(*
  Mark camera system on WEU machine
  1 mark sensor (optional: reverse mode - roll printed in reversed direction, sensor moved to other side)
*)
FUNCTION_BLOCK FB_MarkCamera_WEU EXTENDS FB_CameraBase 
VAR_INPUT
END_VAR
VAR
  // config
  _iMarkDefinition          : I_MarkDefinition;
  // helper
  pMark                     : POINTER TO ST_MarkDefinition;
END_VAR

IF NOT _bInitialized THEN RETURN; END_IF

// The detection work is done in FB_CameraDetection
// This FB just uses(receives) the marks from the external implementation
// - Receives events CamTrigger & CamTriggerDone from MarkDetection
// - Get current marks and send them to the iCameraSink

WHILE _iMarkDefinition.nMarksDetected > _nRxCamPoints DO
  
  pMark := _iMarkDefinition.getMark(nIdx:=_nRxCamPoints+1);
  IF pMark <> 0 THEN
    // Send Mark (CamPoint) to CameraSink
    stCamPoint.x_ref := F_MeterToSubPixelReal(  fPosMeter:=pMark^.fPosX                                 (*[m]*)
                                              , fResoSubPx:=UDINT_TO_LREAL(_nPrintUnitResolution));     (*Result should be in pixels*)
    stCamPoint.y_ref := F_MeterToSubPixelReal( fPosMeter:=pMark^.fPosX                                  (*[m]*)
                                              , fResoSubPx:=UDINT_TO_LREAL(_nPrintUnitResolution));     (*Result should be in pixels*)
    stCamPoint.dx    := F_MeterToSubPixelReal( fPosMeter:=pMark^.sState.dx                              (*[m]*)
                                              , fResoSubPx:=UDINT_TO_LREAL(_nPrintUnitResolution));     (*Result should be in pixels*)
    stCamPoint.dy    := F_MeterToSubPixelReal( fPosMeter:=pMark^.sState.dy                              (*[m]*)
                                              , fResoSubPx:=UDINT_TO_LREAL(_nPrintUnitResolution));     (*Result should be in pixels*)
    stCamPoint.valid := pMark^.sState.bSet;
  
    IF _iCameraSink <> 0 THEN
      _iCameraSink.AddCamPoint(sDeformationPoint:=stCamPoint);
    END_IF
    
    _nRxCamPoints := _nRxCamPoints + 1;   // next mark
  END_IF
END_WHILE

METHOD CamTrigger
VAR_INPUT
  bOk             : BOOL;     // trigger is ok
	nPos            : DINT;     // camera triggered position
  nPosDeviation   : DINT;     // camera started deviation
END_VAR
IF NOT _bInitialized THEN RETURN; END_IF

SUPER^.CamTrigger(bOk:=bOk, nPos:=nPos, nPosDeviation:=nPosDeviation);
END_METHOD

METHOD CamTriggerDone
IF NOT _bInitialized THEN RETURN; END_IF

{warning 'Finalize mark handling'}

SUPER^.CamTriggerDone();
END_METHOD

{attribute 'monitoring':='call'}
PROPERTY eCameraMode : E_CameraMode
GET
eCameraMode := _eCameraMode;
IF _eCameraMode = E_CameraMode.Auto THEN
  eCameraMode := E_CameraMode.Live;
END_IF
END_GET
END_PROPERTY

PROPERTY eDeviceType : E_CameraDevice
GET
eDeviceType := E_CameraDevice.PrintMark;
END_GET
END_PROPERTY

METHOD GetCamStatus : BOOL
VAR_OUTPUT
  bConnectionOK  : BOOL;    // Camera connected
  bTeachOk       : BOOL;    // Teach successful
  nTeachedPoints : UDINT;   // Teached points for this job
  nScannedPoints : UDINT;   // Scanned points on current sheet
  bCamStarted    : BOOL;    // Camera trigger is active, cam started
  bCamDone       : BOOL;    // Camera finished on last CT
  bErrors        : ARRAY[1..GVL_Camera.nC_NbCamErrors] OF BOOL;  // generic error flag list
END_VAR
IF _iMarkDefinition = 0 THEN RETURN; END_IF

bConnectionOK  := TRUE;
bTeachOk       := (_iMarkDefinition.nMarks > 0);
nTeachedPoints := _iMarkDefinition.nMarks;  // teach marks
nScannedPoints := _nRxCamPoints;
bCamStarted    := _bCamTriggerStarted;
bCamDone       := _bCamTriggerDone;

GetCamStatus := bConnectionOK AND bTeachOk;   // camera ready
END_METHOD

METHOD InitMarkCamera
VAR_INPUT
  nPrintUnitResolution         : UDINT;    (*printhead pixel resolution [dpi]*)
  nPrintUnitSubPx              : UDINT;    (*print unit subPixel resolution [SubPx]*)
  iCameraTrigger               : I_CameraTrigger;
  iMarkDefinition              : I_MarkDefinition;  // mark detection fb
END_VAR
VAR
  bOK : BOOL;
END_VAR
SUPER^.Init( nPrintUnitResolution      := nPrintUnitResolution
           , nPrintUnitSubPx           := nPrintUnitSubPx
           , iCameraTrigger            := iCameraTrigger
           , bUseCameraTrigger         := FALSE
           , bUseCameraTriggerFeedback := FALSE);

IF NOT _bInitialized OR iMarkDefinition = 0 THEN LogError('Init: invalid parameter'); RETURN; END_IF

_iMarkDefinition := iMarkDefinition;

_bInitialized := TRUE;
END_METHOD

METHOD mJobStart : BOOL
IF eCameraMode <> E_CameraMode.NoCorrection THEN TeachMarks(); END_IF
END_METHOD

(*
  Set mode to camera.
  :return: TRUE if success
*)
METHOD setCameraMode : BOOL
VAR_INPUT
  eCameraMode : E_CameraMode;
END_VAR
IF eCameraMode = E_CameraMode.Auto OR
   eCameraMode = E_CameraMode.NoCorrection OR
   eCameraMode = E_CameraMode.Live
   //eCameraMode = E_CameraMode.Trend 
THEN
   
  _eCameraMode := eCameraMode;  // set desired mode
  setCameraMode := TRUE;
ELSE
  LogError(F_Concat3('Camera mode=', TO_STRING(eCameraMode), ' not supported by camera'));
  _eCameraMode := E_CameraMode.NoCorrection;
END_IF
END_METHOD

{attribute 'monitoring':='variable'}
PROPERTY sName : STRING
GET
sName := 'Printmarks';
END_GET
END_PROPERTY

(*
  Calculate marks (position, shape) and register to mark definition. 
*)
METHOD PUBLIC TeachMarks : BOOL
VAR_INPUT
END_VAR
VAR
  i : UDINT;
  spacing : LREAL := 0.08;  // mark spacing
  asq : LREAL := 0.002;     // sqare a length
  atr : LREAL := 0.008;     // triangle length (same h / l)
  numMarks : UDINT;
  xOfs : LREAL := 0.0023;
  yOfs : LREAL := 0.0023;
  
  sNewMark : ST_MarkDefinition;
END_VAR


// TODO: this is only a reference caluclation for simulation, please adpat after definition by STAG
//       ...
IF _iMarkDefinition = 0 THEN RETURN; END_IF

_iMarkDefinition.ResetDefinition();

numMarks := TO_UDINT((_fSubstrateLength-2*xOfs) / spacing); //  // TO_UDINT(FLOOR(_fSubstrateLength / spacing);)
IF numMarks = 0 THEN numMarks := 1; END_IF   // at least one mark

// calculate position
FOR i:=1 TO numMarks DO
  sNewMark.fHeight := atr;
  sNewMark.fTrLength := atr;
  sNewMark.fSqLength := SEL(i>1, asq+1.5*atr, asq);
  sNewMark.fPosX := xOfs+(i-1)*spacing;
  sNewMark.fPosY := yOfs;
  sNewMark.bInvertedX := FALSE;
  
  _iMarkDefinition.RegisterMark(sMark:=sNewMark);
END_FOR
END_METHOD

END_FUNCTION_BLOCK

(* stored: Version 1.1.0.1, ProductVersion 3.1.4024.11
   POU FB_MarkCamera_WEU: Id {022ae170-1450-4de8-9411-2fff24170cee}, SpecialFunc None
   Folder I_CameraTriggerDevice: Id {e2dec33a-897c-4e22-aee9-eb47423f04d4}
   Folder Teaching: Id {9779439f-9901-4ac8-a24c-59c2e2c44f9c}
   Method CamTrigger: Id {81474d5d-5e6e-4c16-a459-3afa624802bf}
   Method CamTriggerDone: Id {1b47eb14-3697-493b-9422-5ad8294365cf}
   Property eCameraMode: Id {139b08ce-f2ab-437d-89d4-90989524dcb9}
   Get Get: Id {dcc67e1c-1172-4dc0-8760-a7217421172f}
   Property eDeviceType: Id {4cff99ca-d815-47ed-86bc-fb84d5e4b780}
   Get Get: Id {8d2ae920-228a-44ba-8a46-8bca4ae49bf1}
   Method GetCamStatus: Id {7171f1e1-2bc1-4049-86ae-30de97569022}
   Method InitMarkCamera: Id {0c1aea82-d580-47e9-b922-45dcb8adc4f9}
   Method mJobStart: Id {98df1aac-712b-40bf-ae2a-5c3a55b04142}
   Method setCameraMode: Id {b544e398-6fa9-48f7-9517-2291b5b5ae0e}
   Property sName: Id {19c5cb89-f3d7-4de6-8450-7cd468806f5b}
   Get Get: Id {73270a0c-f7e1-4ad6-9e4c-06f03f404132}
   Method TeachMarks: Id {bda865f2-b959-47c0-bd1d-61d48f369350} *)
